{attribute 'GeneratedUsingTerminal: EK1960-2600-0019'}
{attribute addProperty BoxType "EK1960-2600-0019"}
{attribute addProperty Id "FSoE_CommandUSINT1FSOUT_Module_1_Module_FaultBOOL1FSOUT_Module_2_Module_FaultBOOL1FSOUT_Module_3_Module_FaultBOOL1FSOUT_Module_4_Module_FaultBOOL1FSOUT_Module_5_Module_FaultBOOL1FSOUT_Module_6_Module_FaultBOOL1FSOUT_Relais_Module_Module_FaultBOOL1FSIN_Module_1_Channel_1_InputBOOL1FSIN_Module_1_Channel_2_InputBOOL1FSIN_Module_1_Module_FaultBOOL1FSIN_Module_2_Channel_1_InputBOOL1FSIN_Module_2_Channel_2_InputBOOL1FSIN_Module_2_Module_FaultBOOL1FSIN_Module_3_Channel_1_InputBOOL1FSIN_Module_3_Channel_2_InputBOOL1FSIN_Module_3_Module_FaultBOOL1FSoE_CRC_000UINT2FSIN_Module_4_Channel_1_InputBOOL1FSIN_Module_4_Channel_2_InputBOOL1FSIN_Module_4_Module_FaultBOOL1FSIN_Module_5_Channel_1_InputBOOL1FSIN_Module_5_Channel_2_InputBOOL1FSIN_Module_5_Module_FaultBOOL1FSIN_Module_6_Channel_1_InputBOOL1FSIN_Module_6_Channel_2_InputBOOL1FSIN_Module_6_Module_FaultBOOL1FSIN_Module_7_Channel_1_InputBOOL1FSIN_Module_7_Channel_2_InputBOOL1FSIN_Module_7_Module_FaultBOOL1FSIN_Module_8_Channel_1_InputBOOL1FSIN_Module_8_Channel_2_InputBOOL1FSIN_Module_8_Module_FaultBOOL1FSIN_Module_9_Channel_1_InputBOOL1FSoE_CRC_001UINT2FSIN_Module_9_Channel_2_InputBOOL1FSIN_Module_9_Module_Fault_1BOOL1FSIN_Module_9_Module_Fault_2BOOL1FSIN_Module_10_Channel_1_InputBOOL1FSIN_Module_10_Channel_2_InputBOOL1FSIN_Module_10_Module_Fault_1BOOL1FSIN_Module_10_Module_Fault_2BOOL1FSoE_CRC_002UINT2FSoE_Connection_IDUINT2"}
{attribute addProperty CRC "3131524987"}
{attribute addProperty Size "48"}
TYPE FSOE_BAA7477B :
STRUCT
	{attribute addProperty Name "FSoE_Command"}
	FSoE_Command : USINT;
	{attribute addProperty Name "FSOUT_Module_1_Module_Fault"}
	FSOUT_Module_1_Module_Fault : BOOL;
	{attribute addProperty Name "FSOUT_Module_2_Module_Fault"}
	FSOUT_Module_2_Module_Fault : BOOL;
	{attribute addProperty Name "FSOUT_Module_3_Module_Fault"}
	FSOUT_Module_3_Module_Fault : BOOL;
	{attribute addProperty Name "FSOUT_Module_4_Module_Fault"}
	FSOUT_Module_4_Module_Fault : BOOL;
	{attribute addProperty Name "FSOUT_Module_5_Module_Fault"}
	FSOUT_Module_5_Module_Fault : BOOL;
	{attribute addProperty Name "FSOUT_Module_6_Module_Fault"}
	FSOUT_Module_6_Module_Fault : BOOL;
	{attribute addProperty Name "FSOUT_Relais_Module_Module_Fault"}
	FSOUT_Relais_Module_Module_Fault : BOOL;
	{attribute addProperty Name "FSIN_Module_1_Channel_1_Input"}
	FSIN_Module_1_Channel_1_Input : BOOL;
	{attribute addProperty Name "FSIN_Module_1_Channel_2_Input"}
	FSIN_Module_1_Channel_2_Input : BOOL;
	{attribute addProperty Name "FSIN_Module_1_Module_Fault"}
	FSIN_Module_1_Module_Fault : BOOL;
	{attribute addProperty Name "FSIN_Module_2_Channel_1_Input"}
	FSIN_Module_2_Channel_1_Input : BOOL;
	{attribute addProperty Name "FSIN_Module_2_Channel_2_Input"}
	FSIN_Module_2_Channel_2_Input : BOOL;
	{attribute addProperty Name "FSIN_Module_2_Module_Fault"}
	FSIN_Module_2_Module_Fault : BOOL;
	{attribute addProperty Name "FSIN_Module_3_Channel_1_Input"}
	FSIN_Module_3_Channel_1_Input : BOOL;
	{attribute addProperty Name "FSIN_Module_3_Channel_2_Input"}
	FSIN_Module_3_Channel_2_Input : BOOL;
	{attribute addProperty Name "FSIN_Module_3_Module_Fault"}
	FSIN_Module_3_Module_Fault : BOOL;
	{attribute addProperty Name "FSoE_CRC_000"}
	FSoE_CRC_000 : UINT;
	{attribute addProperty Name "FSIN_Module_4_Channel_1_Input"}
	FSIN_Module_4_Channel_1_Input : BOOL;
	{attribute addProperty Name "FSIN_Module_4_Channel_2_Input"}
	FSIN_Module_4_Channel_2_Input : BOOL;
	{attribute addProperty Name "FSIN_Module_4_Module_Fault"}
	FSIN_Module_4_Module_Fault : BOOL;
	{attribute addProperty Name "FSIN_Module_5_Channel_1_Input"}
	FSIN_Module_5_Channel_1_Input : BOOL;
	{attribute addProperty Name "FSIN_Module_5_Channel_2_Input"}
	FSIN_Module_5_Channel_2_Input : BOOL;
	{attribute addProperty Name "FSIN_Module_5_Module_Fault"}
	FSIN_Module_5_Module_Fault : BOOL;
	{attribute addProperty Name "FSIN_Module_6_Channel_1_Input"}
	FSIN_Module_6_Channel_1_Input : BOOL;
	{attribute addProperty Name "FSIN_Module_6_Channel_2_Input"}
	FSIN_Module_6_Channel_2_Input : BOOL;
	{attribute addProperty Name "FSIN_Module_6_Module_Fault"}
	FSIN_Module_6_Module_Fault : BOOL;
	{attribute addProperty Name "FSIN_Module_7_Channel_1_Input"}
	FSIN_Module_7_Channel_1_Input : BOOL;
	{attribute addProperty Name "FSIN_Module_7_Channel_2_Input"}
	FSIN_Module_7_Channel_2_Input : BOOL;
	{attribute addProperty Name "FSIN_Module_7_Module_Fault"}
	FSIN_Module_7_Module_Fault : BOOL;
	{attribute addProperty Name "FSIN_Module_8_Channel_1_Input"}
	FSIN_Module_8_Channel_1_Input : BOOL;
	{attribute addProperty Name "FSIN_Module_8_Channel_2_Input"}
	FSIN_Module_8_Channel_2_Input : BOOL;
	{attribute addProperty Name "FSIN_Module_8_Module_Fault"}
	FSIN_Module_8_Module_Fault : BOOL;
	{attribute addProperty Name "FSIN_Module_9_Channel_1_Input"}
	FSIN_Module_9_Channel_1_Input : BOOL;
	{attribute addProperty Name "FSoE_CRC_001"}
	FSoE_CRC_001 : UINT;
	{attribute addProperty Name "FSIN_Module_9_Channel_2_Input"}
	FSIN_Module_9_Channel_2_Input : BOOL;
	{attribute addProperty Name "FSIN_Module_9_Module_Fault_1"}
	FSIN_Module_9_Module_Fault_1 : BOOL;
	{attribute addProperty Name "FSIN_Module_9_Module_Fault_2"}
	FSIN_Module_9_Module_Fault_2 : BOOL;
	{attribute addProperty Name "FSIN_Module_10_Channel_1_Input"}
	FSIN_Module_10_Channel_1_Input : BOOL;
	{attribute addProperty Name "FSIN_Module_10_Channel_2_Input"}
	FSIN_Module_10_Channel_2_Input : BOOL;
	{attribute addProperty Name "FSIN_Module_10_Module_Fault_1"}
	FSIN_Module_10_Module_Fault_1 : BOOL;
	{attribute addProperty Name "FSIN_Module_10_Module_Fault_2"}
	FSIN_Module_10_Module_Fault_2 : BOOL;
	{attribute addProperty Name "FSoE_CRC_002"}
	FSoE_CRC_002 : UINT;
	{attribute addProperty Name "FSoE_Connection_ID"}
	FSoE_Connection_ID : UINT;
END_STRUCT
END_TYPE

(* stored: Version 1.2.0.0, ProductVersion 3.1.4024.9
   DUT FSOE_BAA7477B: Id {0c2c38b5-9758-4393-92ee-dc0b3442d290} *)
